(* Logix 5000 project; controller SX_V040001_C001 vendor 1 type 14 code 77 rev 16.23; software revision 16.04; part 2 of 35 *)
(* tags used below, declared in another part *)
   ALARM_BITS : INT[10];
   ALL_KINDS : INT[90];
   Basic : INT;
   CMD : INT[36];
   DRIVE : INT[32];
   EMPTYING : INT[18];
   FP_ALARM_RESET : BOOL;
   G_DInput : DINT[3];
   G_DOutput : DINT[3];
   loading : INT[19];
   louvre : INT[11];
   m_alarm_exist : BOOL;
   m_alarm_horn : BOOL;
   m_element_fault_reset : BOOL;
   m_notstop : BOOL;
   m_on_off_line : BOOL;
   m_power_up : BOOL;
   METERING : INT[44];
   mw_major_fault : DINT;
   PARAMETER : INT[501];
   T_MAX_CURRENT : TIMER;
   T_SCRAPER : TIMER;
   T_START_ALARM : TIMER;
   TEMP : INT[14];
   Z15 : COUNTER;
   Z16 : COUNTER;
   Z17 : COUNTER;
   Z18 : COUNTER;
   Z19 : COUNTER;
   Z20 : COUNTER;
   Z21 : COUNTER;
   Z22 : COUNTER;
   Z23 : COUNTER;
   Z24 : COUNTER;
   Z25 : COUNTER;
   Z26 : COUNTER;
   Z27 : COUNTER;
   Z28 : COUNTER;
   Z29 : COUNTER;
   Z30 : COUNTER;
   Z31 : COUNTER;
   Z32 : COUNTER;
   Z33 : COUNTER;
   Z34 : COUNTER;
   Z35 : COUNTER;
   Z36 : COUNTER;
   Z37 : COUNTER;
   Z38 : COUNTER;
   Z39 : COUNTER;
   Z40 : COUNTER;
   Z41 : COUNTER;
   Z42 : COUNTER;
   Z43 : COUNTER;
   Z44 : COUNTER;
   Z45 : COUNTER;
   Z46 : COUNTER;
   Z47 : COUNTER;
   Z48 : COUNTER;
   Z49 : COUNTER;
   Z50 : COUNTER;
(* MainProgram, continued *)

ROUTINE Alarms   (* ladder *)
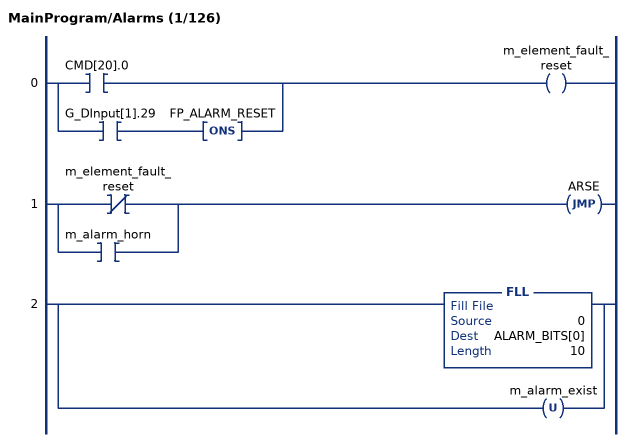
   0: [XIC(CMD[20].0) ,XIC(G_DInput[1].29) ONS(FP_ALARM_RESET) ]OTE(m_element_fault_reset);
   1: [XIO(m_element_fault_reset) ,XIC(m_alarm_horn) ]JMP(ARSE);
   2: [FLL(0,ALARM_BITS[0],10) ,OTU(m_alarm_exist) ];
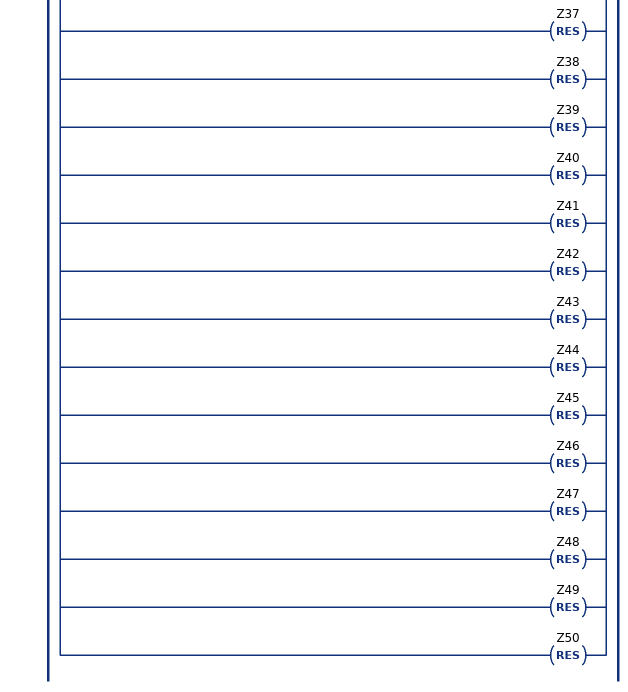
   3: [RES(Z15) ,RES(Z16) ,RES(Z17) ,RES(Z18) ,RES(Z19) ,RES(Z20) ,RES(Z21) ,RES(Z22) ,RES(Z23) ,RES(Z24) ,RES(Z25) ,RES(Z26) ,RES(Z27) ,RES(Z28) ,RES(Z29) ,RES(Z30) ,RES(Z31) ,RES(Z32) ,RES(Z33) ,RES(Z34) ,RES(Z35) ,RES(Z36) ,RES(Z37) ,RES(Z38) ,RES(Z39) ,RES(Z40) ,RES(Z41) ,RES(Z42) ,RES(Z43) ,RES(Z44) ,RES(Z45) ,RES(Z46) ,RES(Z47) ,RES(Z48) ,RES(Z49) ,RES(Z50) ];
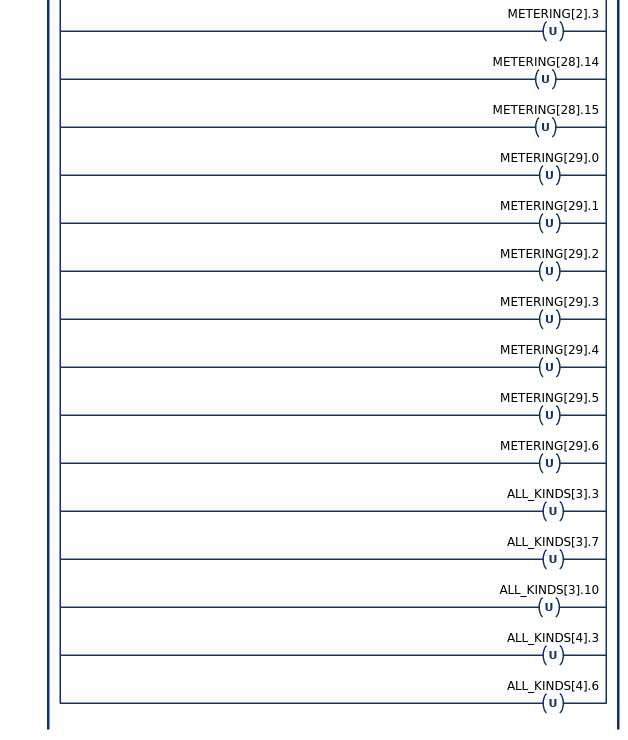
   4: [OTU(TEMP[1].0) ,OTU(TEMP[1].1) ,OTU(TEMP[1].3) ,OTU(TEMP[1].5) ,OTU(TEMP[1].6) ,OTU(DRIVE[2].8) ,OTU(DRIVE[2].9) ,OTU(DRIVE[2].10) ,OTU(DRIVE[2].11) ,OTU(EMPTYING[1].5) ,OTU(EMPTYING[1].7) ,OTU(EMPTYING[1].8) ,OTU(EMPTYING[1].11) ,OTU(EMPTYING[1].12) ,OTU(loading[2].0) ,OTU(loading[2].1) ,OTU(louvre[3].10) ,OTU(louvre[4].10) ,OTU(METERING[1].15) ,OTU(METERING[2].0) ,OTU(METERING[2].1) ,OTU(METERING[2].2) ,OTU(METERING[2].3) ,OTU(METERING[28].14) ,OTU(METERING[28].15) ,OTU(METERING[29].0) ,OTU(METERING[29].1) ,OTU(METERING[29].2) ,OTU(METERING[29].3) ,OTU(METERING[29].4) ,OTU(METERING[29].5) ,OTU(METERING[29].6) ,OTU(ALL_KINDS[3].3) ,OTU(ALL_KINDS[3].7) ,OTU(ALL_KINDS[3].10) ,OTU(ALL_KINDS[4].3) ,OTU(ALL_KINDS[4].6) ];
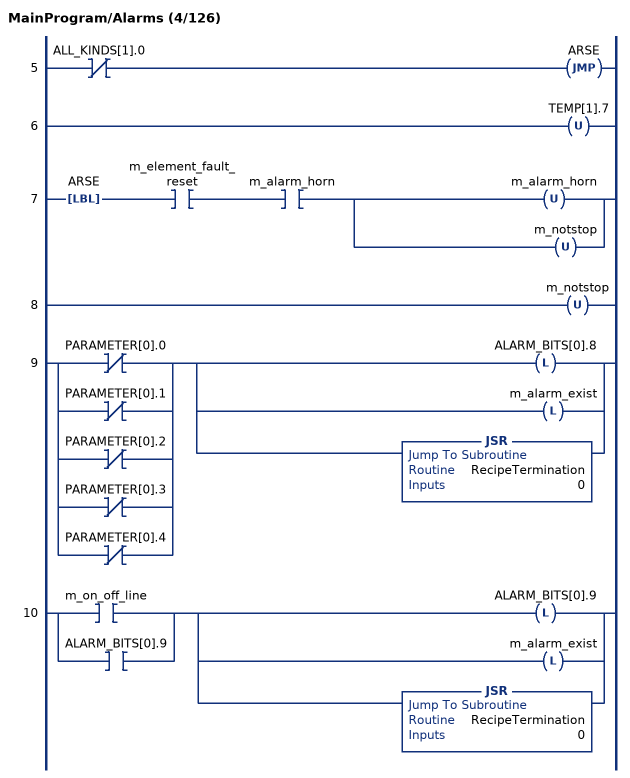
   5: XIO(ALL_KINDS[1].0)JMP(ARSE);
   6: OTU(TEMP[1].7);
   7: LBL(ARSE)XIC(m_element_fault_reset)XIC(m_alarm_horn)[OTU(m_alarm_horn) ,OTU(m_notstop) ];
   8: OTU(m_notstop);
   9: [XIO(PARAMETER[0].0) ,XIO(PARAMETER[0].1) ,XIO(PARAMETER[0].2) ,XIO(PARAMETER[0].3) ,XIO(PARAMETER[0].4) ][OTL(ALARM_BITS[0].8) ,OTL(m_alarm_exist) ,JSR(RecipeTermination,0) ];
   10: [XIC(m_on_off_line) ,XIC(ALARM_BITS[0].9) ][OTL(ALARM_BITS[0].9) ,OTL(m_alarm_exist) ,JSR(RecipeTermination,0) ];
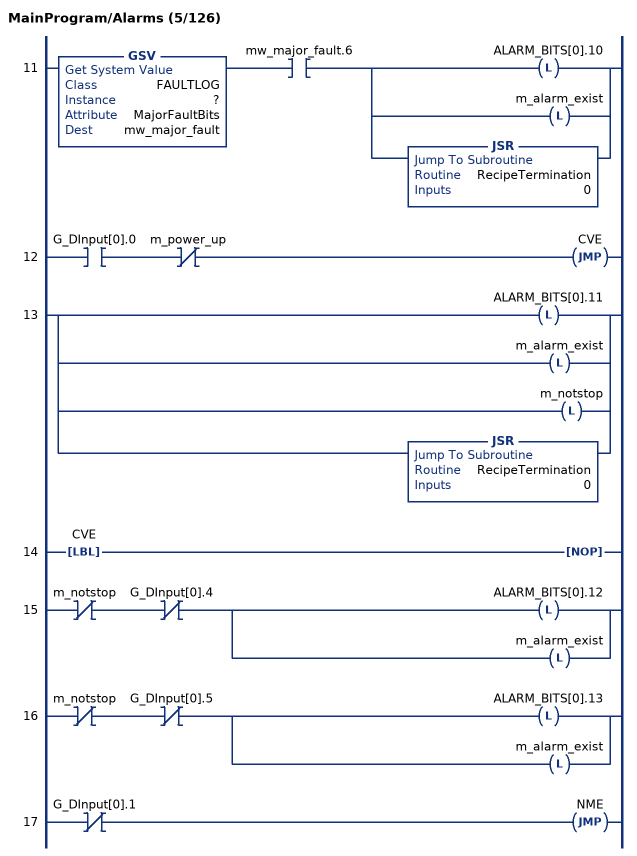
   11: GSV(FAULTLOG,?,MajorFaultBits,mw_major_fault)XIC(mw_major_fault.6)[OTL(ALARM_BITS[0].10) ,OTL(m_alarm_exist) ,JSR(RecipeTermination,0) ];
   12: XIC(G_DInput[0].0)XIO(m_power_up)JMP(CVE);
   13: [OTL(ALARM_BITS[0].11) ,OTL(m_alarm_exist) ,OTL(m_notstop) ,JSR(RecipeTermination,0) ];
   14: LBL(CVE)NOP();
   15: XIO(m_notstop)XIO(G_DInput[0].4)[OTL(ALARM_BITS[0].12) ,OTL(m_alarm_exist) ];
   16: XIO(m_notstop)XIO(G_DInput[0].5)[OTL(ALARM_BITS[0].13) ,OTL(m_alarm_exist) ];
   17: XIO(G_DInput[0].1)JMP(NME);
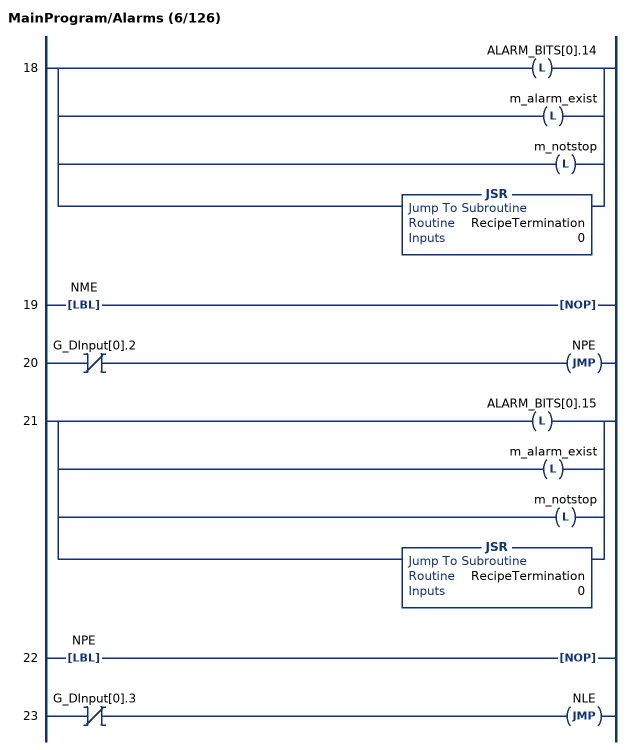
   18: [OTL(ALARM_BITS[0].14) ,OTL(m_alarm_exist) ,OTL(m_notstop) ,JSR(RecipeTermination,0) ];
   19: LBL(NME)NOP();
   20: XIO(G_DInput[0].2)JMP(NPE);
   21: [OTL(ALARM_BITS[0].15) ,OTL(m_alarm_exist) ,OTL(m_notstop) ,JSR(RecipeTermination,0) ];
   22: LBL(NPE)NOP();
   23: XIO(G_DInput[0].3)JMP(NLE);
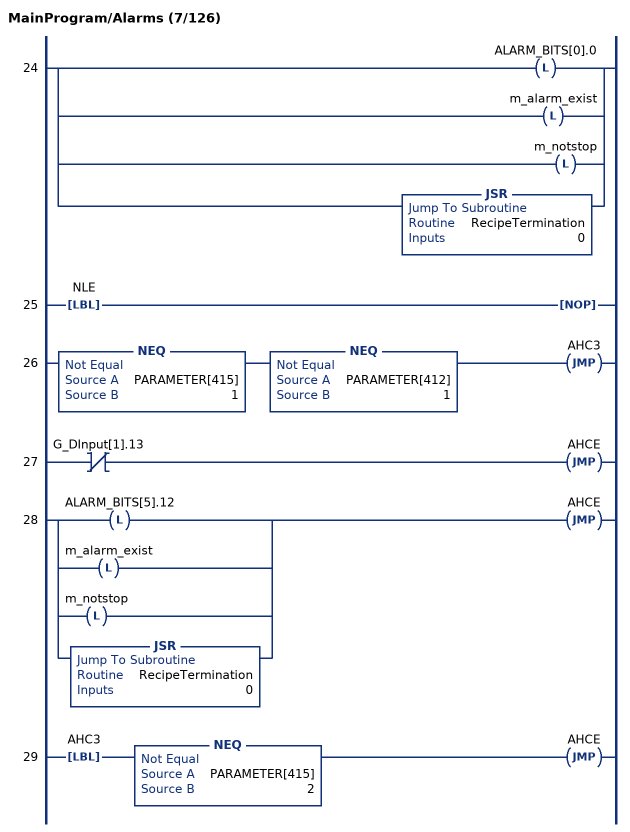
   24: [OTL(ALARM_BITS[0].0) ,OTL(m_alarm_exist) ,OTL(m_notstop) ,JSR(RecipeTermination,0) ];
   25: LBL(NLE)NOP();
   26: NEQ(PARAMETER[415],1)NEQ(PARAMETER[412],1)JMP(AHC3);
   27: XIO(G_DInput[1].13)JMP(AHCE);
   28: [OTL(ALARM_BITS[5].12) ,OTL(m_alarm_exist) ,OTL(m_notstop) ,JSR(RecipeTermination,0) ]JMP(AHCE);
   29: LBL(AHC3)NEQ(PARAMETER[415],2)JMP(AHCE);
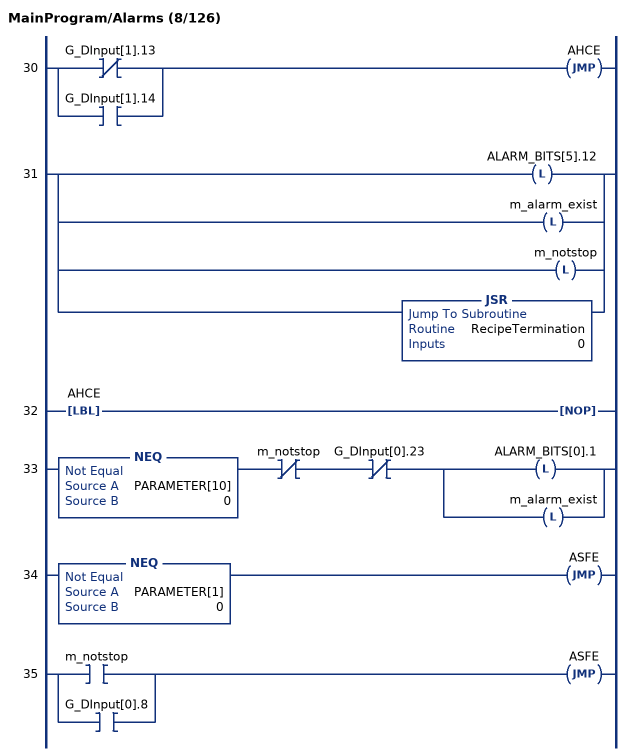
   30: [XIO(G_DInput[1].13) ,XIC(G_DInput[1].14) ]JMP(AHCE);
   31: [OTL(ALARM_BITS[5].12) ,OTL(m_alarm_exist) ,OTL(m_notstop) ,JSR(RecipeTermination,0) ];
   32: LBL(AHCE)NOP();
   33: NEQ(PARAMETER[10],0)XIO(m_notstop)XIO(G_DInput[0].23)[OTL(ALARM_BITS[0].1) ,OTL(m_alarm_exist) ];
   34: NEQ(PARAMETER[1],0)JMP(ASFE);
   35: [XIC(m_notstop) ,XIC(G_DInput[0].8) ]JMP(ASFE);
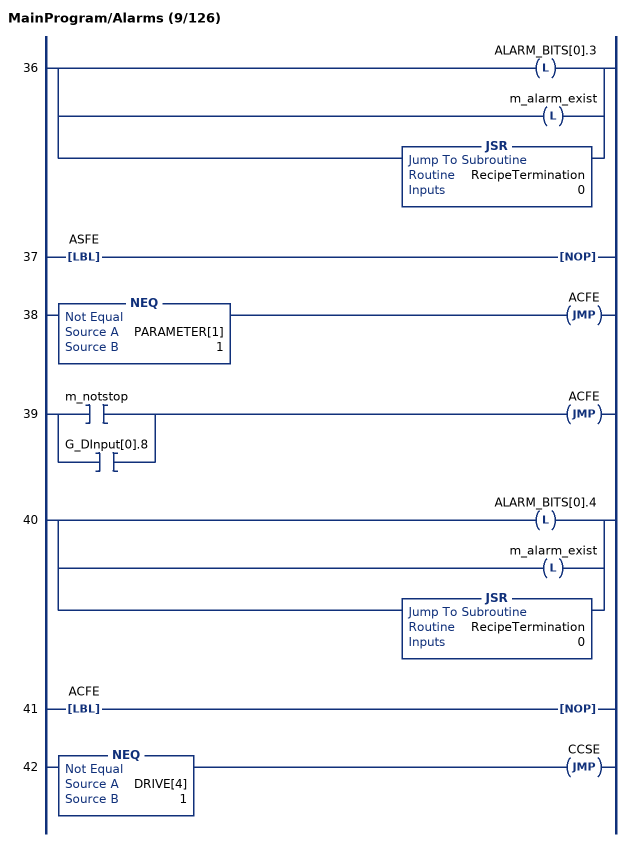
   36: [OTL(ALARM_BITS[0].3) ,OTL(m_alarm_exist) ,JSR(RecipeTermination,0) ];
   37: LBL(ASFE)NOP();
   38: NEQ(PARAMETER[1],1)JMP(ACFE);
   39: [XIC(m_notstop) ,XIC(G_DInput[0].8) ]JMP(ACFE);
   40: [OTL(ALARM_BITS[0].4) ,OTL(m_alarm_exist) ,JSR(RecipeTermination,0) ];
   41: LBL(ACFE)NOP();
   42: NEQ(DRIVE[4],1)JMP(CCSE);
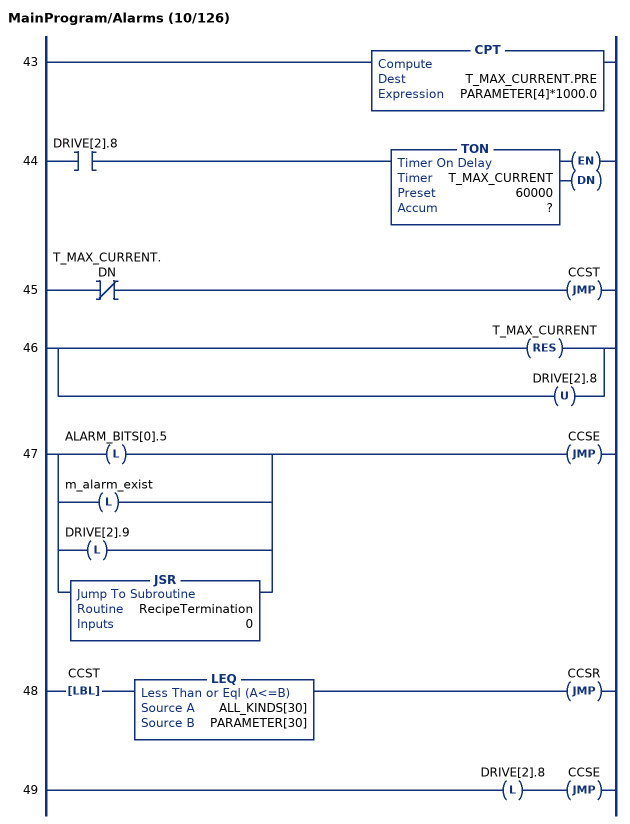
   43: CPT(T_MAX_CURRENT.PRE,PARAMETER[4]*1000.0);
   44: XIC(DRIVE[2].8)TON(T_MAX_CURRENT,?,?);
   45: XIO(T_MAX_CURRENT.DN)JMP(CCST);
   46: [RES(T_MAX_CURRENT) ,OTU(DRIVE[2].8) ];
   47: [OTL(ALARM_BITS[0].5) ,OTL(m_alarm_exist) ,OTL(DRIVE[2].9) ,JSR(RecipeTermination,0) ]JMP(CCSE);
   48: LBL(CCST)LEQ(ALL_KINDS[30],PARAMETER[30])JMP(CCSR);
   49: OTL(DRIVE[2].8)JMP(CCSE);
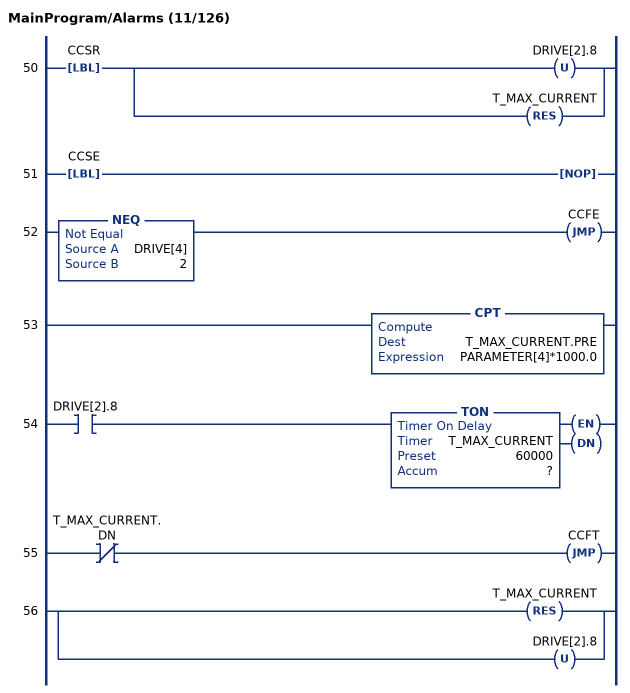
   50: LBL(CCSR)[OTU(DRIVE[2].8) ,RES(T_MAX_CURRENT) ];
   51: LBL(CCSE)NOP();
   52: NEQ(DRIVE[4],2)JMP(CCFE);
   53: CPT(T_MAX_CURRENT.PRE,PARAMETER[4]*1000.0);
   54: XIC(DRIVE[2].8)TON(T_MAX_CURRENT,?,?);
   55: XIO(T_MAX_CURRENT.DN)JMP(CCFT);
   56: [RES(T_MAX_CURRENT) ,OTU(DRIVE[2].8) ];
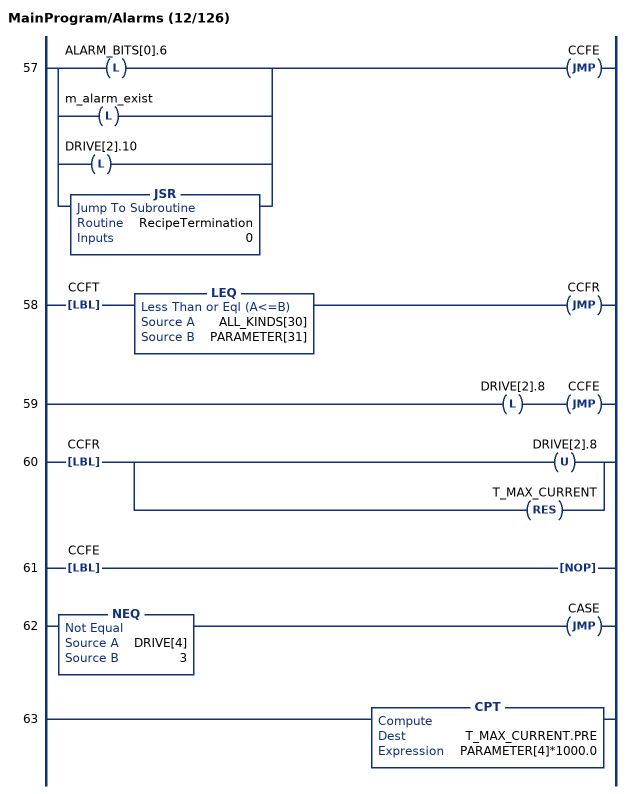
   57: [OTL(ALARM_BITS[0].6) ,OTL(m_alarm_exist) ,OTL(DRIVE[2].10) ,JSR(RecipeTermination,0) ]JMP(CCFE);
   58: LBL(CCFT)LEQ(ALL_KINDS[30],PARAMETER[31])JMP(CCFR);
   59: OTL(DRIVE[2].8)JMP(CCFE);
   60: LBL(CCFR)[OTU(DRIVE[2].8) ,RES(T_MAX_CURRENT) ];
   61: LBL(CCFE)NOP();
   62: NEQ(DRIVE[4],3)JMP(CASE);
   63: CPT(T_MAX_CURRENT.PRE,PARAMETER[4]*1000.0);
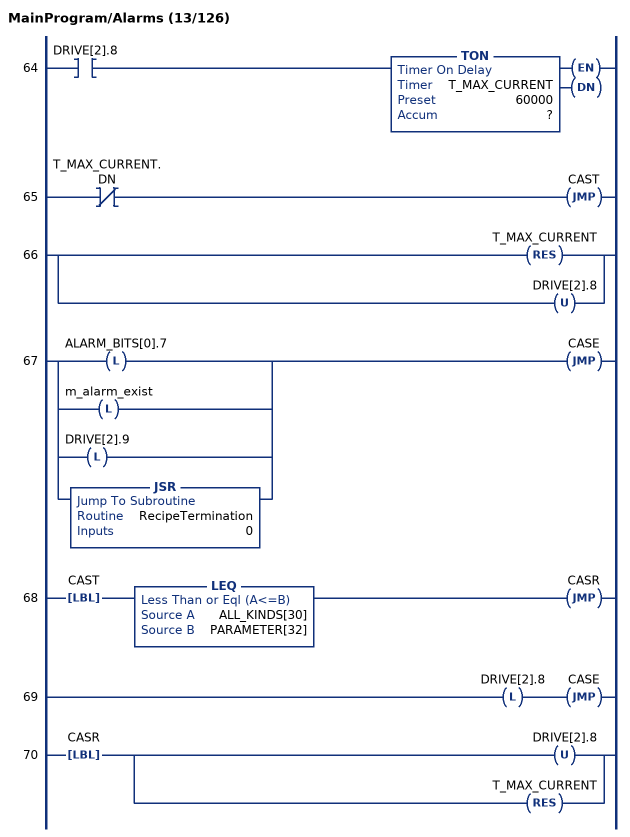
   64: XIC(DRIVE[2].8)TON(T_MAX_CURRENT,?,?);
   65: XIO(T_MAX_CURRENT.DN)JMP(CAST);
   66: [RES(T_MAX_CURRENT) ,OTU(DRIVE[2].8) ];
   67: [OTL(ALARM_BITS[0].7) ,OTL(m_alarm_exist) ,OTL(DRIVE[2].9) ,JSR(RecipeTermination,0) ]JMP(CASE);
   68: LBL(CAST)LEQ(ALL_KINDS[30],PARAMETER[32])JMP(CASR);
   69: OTL(DRIVE[2].8)JMP(CASE);
   70: LBL(CASR)[OTU(DRIVE[2].8) ,RES(T_MAX_CURRENT) ];
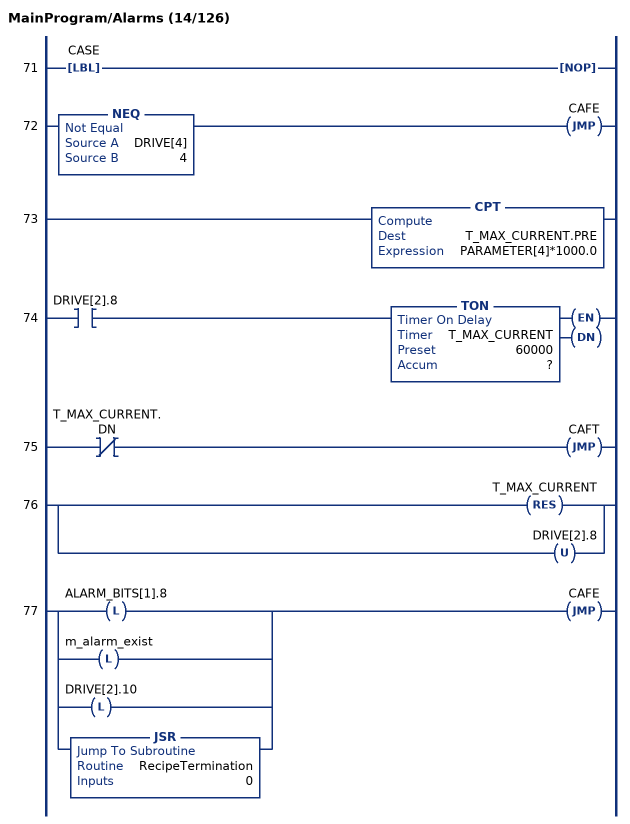
   71: LBL(CASE)NOP();
   72: NEQ(DRIVE[4],4)JMP(CAFE);
   73: CPT(T_MAX_CURRENT.PRE,PARAMETER[4]*1000.0);
   74: XIC(DRIVE[2].8)TON(T_MAX_CURRENT,?,?);
   75: XIO(T_MAX_CURRENT.DN)JMP(CAFT);
   76: [RES(T_MAX_CURRENT) ,OTU(DRIVE[2].8) ];
   77: [OTL(ALARM_BITS[1].8) ,OTL(m_alarm_exist) ,OTL(DRIVE[2].10) ,JSR(RecipeTermination,0) ]JMP(CAFE);
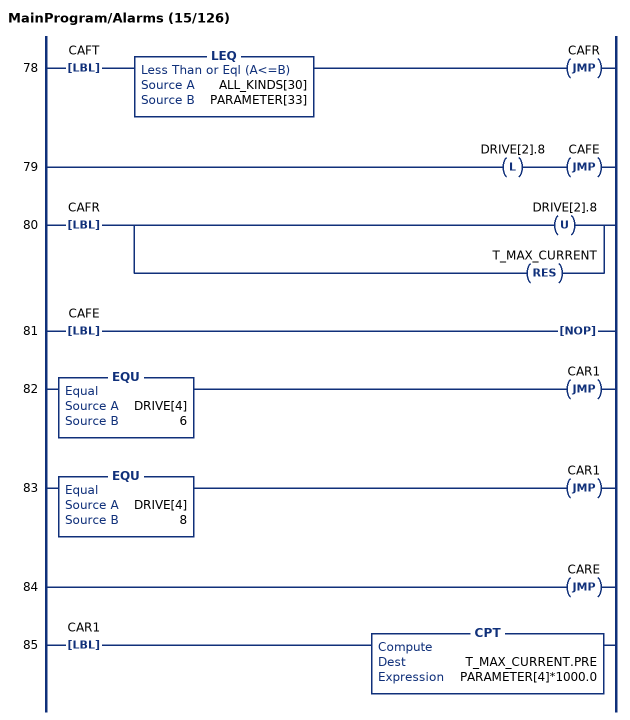
   78: LBL(CAFT)LEQ(ALL_KINDS[30],PARAMETER[33])JMP(CAFR);
   79: OTL(DRIVE[2].8)JMP(CAFE);
   80: LBL(CAFR)[OTU(DRIVE[2].8) ,RES(T_MAX_CURRENT) ];
   81: LBL(CAFE)NOP();
   82: EQU(DRIVE[4],6)JMP(CAR1);
   83: EQU(DRIVE[4],8)JMP(CAR1);
   84: JMP(CARE);
   85: LBL(CAR1)CPT(T_MAX_CURRENT.PRE,PARAMETER[4]*1000.0);
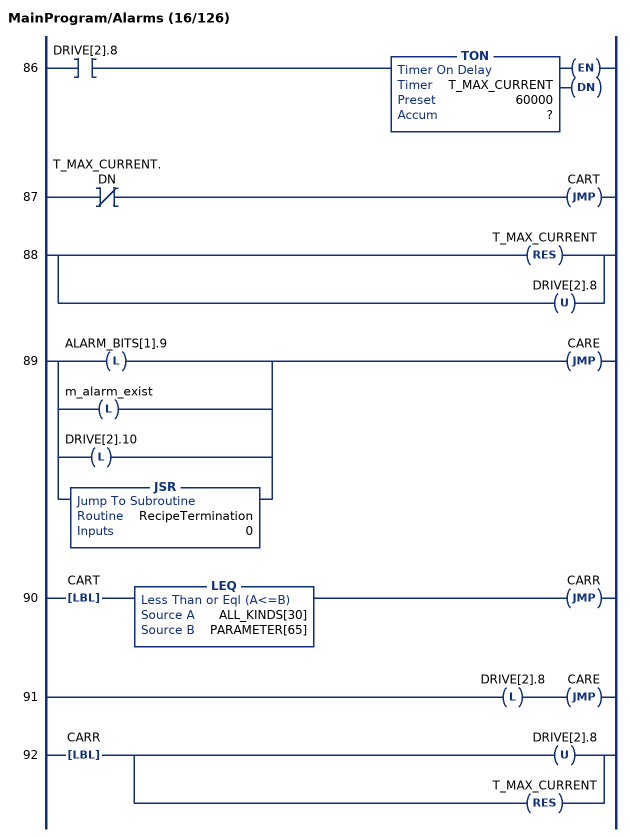
   86: XIC(DRIVE[2].8)TON(T_MAX_CURRENT,?,?);
   87: XIO(T_MAX_CURRENT.DN)JMP(CART);
   88: [RES(T_MAX_CURRENT) ,OTU(DRIVE[2].8) ];
   89: [OTL(ALARM_BITS[1].9) ,OTL(m_alarm_exist) ,OTL(DRIVE[2].10) ,JSR(RecipeTermination,0) ]JMP(CARE);
   90: LBL(CART)LEQ(ALL_KINDS[30],PARAMETER[65])JMP(CARR);
   91: OTL(DRIVE[2].8)JMP(CARE);
   92: LBL(CARR)[OTU(DRIVE[2].8) ,RES(T_MAX_CURRENT) ];
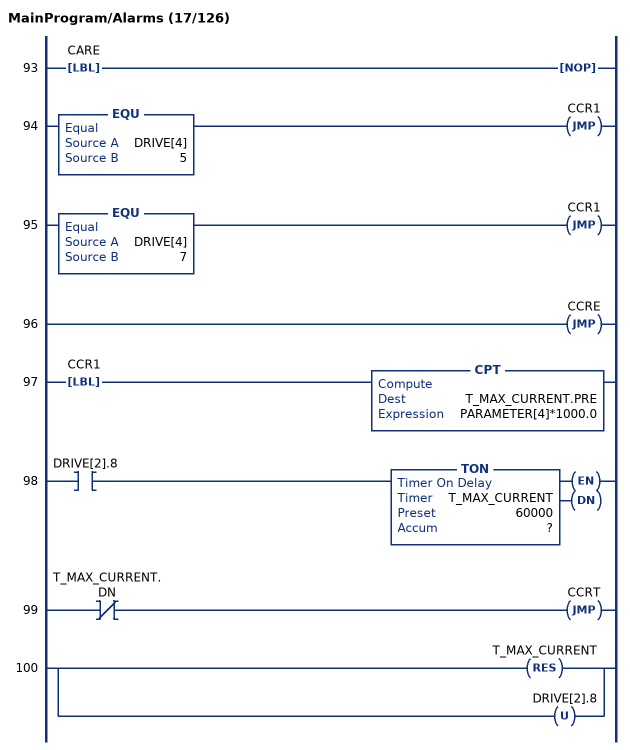
   93: LBL(CARE)NOP();
   94: EQU(DRIVE[4],5)JMP(CCR1);
   95: EQU(DRIVE[4],7)JMP(CCR1);
   96: JMP(CCRE);
   97: LBL(CCR1)CPT(T_MAX_CURRENT.PRE,PARAMETER[4]*1000.0);
   98: XIC(DRIVE[2].8)TON(T_MAX_CURRENT,?,?);
   99: XIO(T_MAX_CURRENT.DN)JMP(CCRT);
   100: [RES(T_MAX_CURRENT) ,OTU(DRIVE[2].8) ];
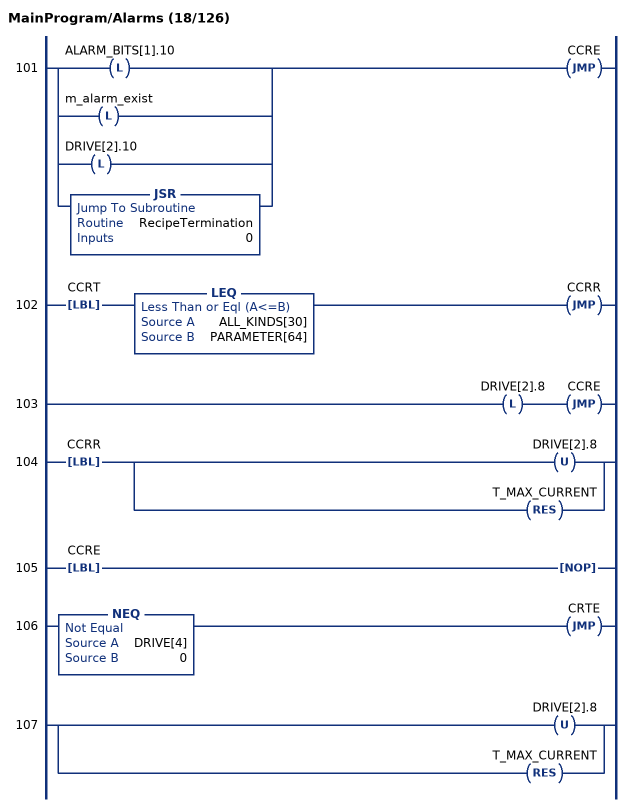
   101: [OTL(ALARM_BITS[1].10) ,OTL(m_alarm_exist) ,OTL(DRIVE[2].10) ,JSR(RecipeTermination,0) ]JMP(CCRE);
   102: LBL(CCRT)LEQ(ALL_KINDS[30],PARAMETER[64])JMP(CCRR);
   103: OTL(DRIVE[2].8)JMP(CCRE);
   104: LBL(CCRR)[OTU(DRIVE[2].8) ,RES(T_MAX_CURRENT) ];
   105: LBL(CCRE)NOP();
   106: NEQ(DRIVE[4],0)JMP(CRTE);
   107: [OTU(DRIVE[2].8) ,RES(T_MAX_CURRENT) ];
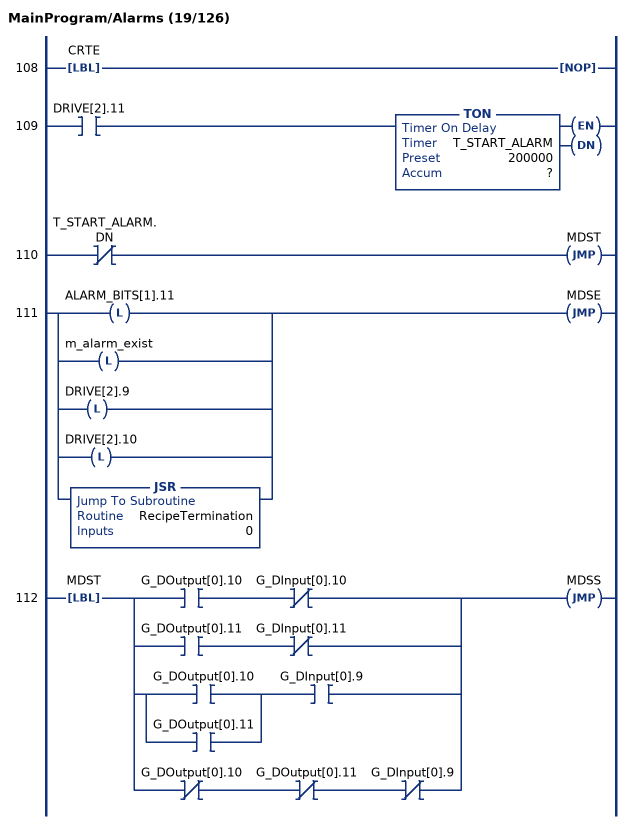
   108: LBL(CRTE)NOP();
   109: XIC(DRIVE[2].11)TON(T_START_ALARM,?,?);
   110: XIO(T_START_ALARM.DN)JMP(MDST);
   111: [OTL(ALARM_BITS[1].11) ,OTL(m_alarm_exist) ,OTL(DRIVE[2].9) ,OTL(DRIVE[2].10) ,JSR(RecipeTermination,0) ]JMP(MDSE);
   112: LBL(MDST)[XIC(G_DOutput[0].10) XIO(G_DInput[0].10) ,XIC(G_DOutput[0].11) XIO(G_DInput[0].11) ,[XIC(G_DOutput[0].10) ,XIC(G_DOutput[0].11) ] XIC(G_DInput[0].9) ,XIO(G_DOutput[0].10) XIO(G_DOutput[0].11) XIO(G_DInput[0].9) ]JMP(MDSS);
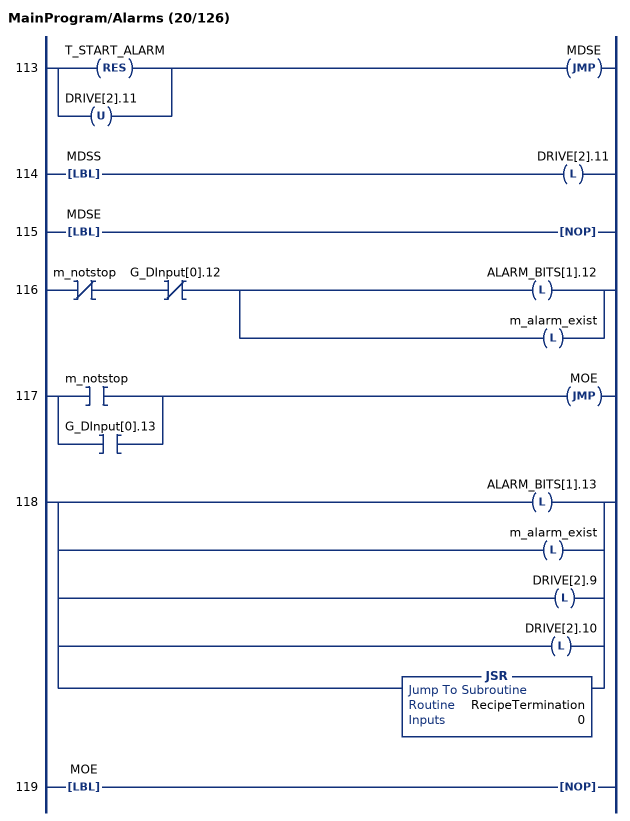
   113: [RES(T_START_ALARM) ,OTU(DRIVE[2].11) ]JMP(MDSE);
   114: LBL(MDSS)OTL(DRIVE[2].11);
   115: LBL(MDSE)NOP();
   116: XIO(m_notstop)XIO(G_DInput[0].12)[OTL(ALARM_BITS[1].12) ,OTL(m_alarm_exist) ];
   117: [XIC(m_notstop) ,XIC(G_DInput[0].13) ]JMP(MOE);
   118: [OTL(ALARM_BITS[1].13) ,OTL(m_alarm_exist) ,OTL(DRIVE[2].9) ,OTL(DRIVE[2].10) ,JSR(RecipeTermination,0) ];
   119: LBL(MOE)NOP();
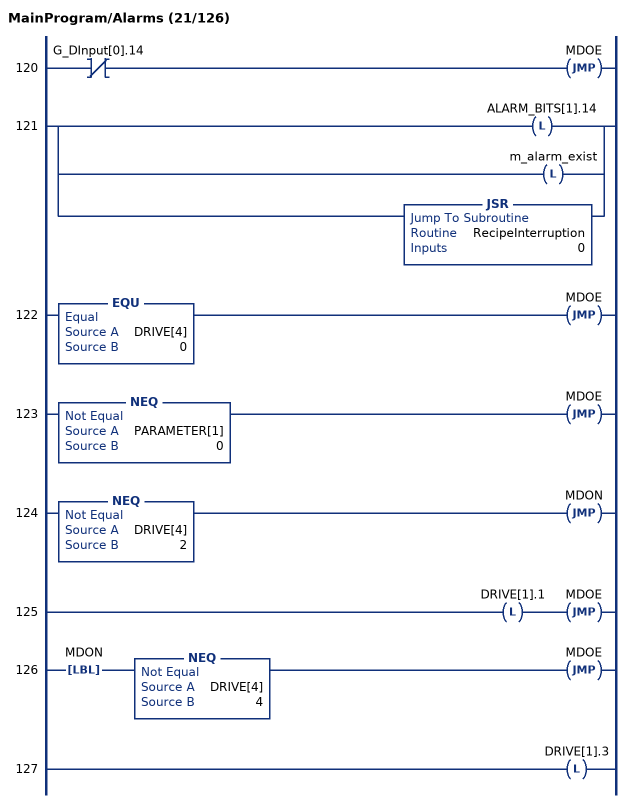
   120: XIO(G_DInput[0].14)JMP(MDOE);
   121: [OTL(ALARM_BITS[1].14) ,OTL(m_alarm_exist) ,JSR(RecipeInterruption,0) ];
   122: EQU(DRIVE[4],0)JMP(MDOE);
   123: NEQ(PARAMETER[1],0)JMP(MDOE);
   124: NEQ(DRIVE[4],2)JMP(MDON);
   125: OTL(DRIVE[1].1)JMP(MDOE);
   126: LBL(MDON)NEQ(DRIVE[4],4)JMP(MDOE);
   127: OTL(DRIVE[1].3);
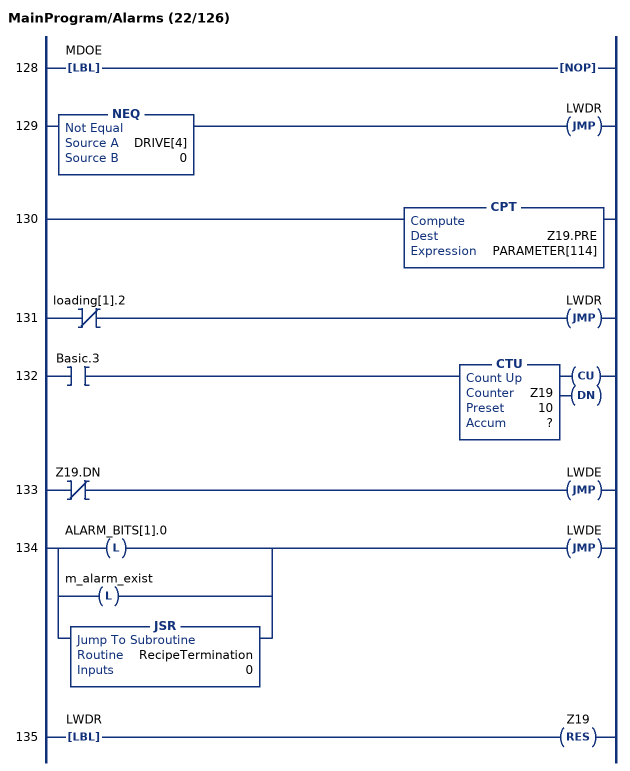
   128: LBL(MDOE)NOP();
   129: NEQ(DRIVE[4],0)JMP(LWDR);
   130: CPT(Z19.PRE,PARAMETER[114]);
   131: XIO(loading[1].2)JMP(LWDR);
   132: XIC(Basic.3)CTU(Z19,?,?);
   133: XIO(Z19.DN)JMP(LWDE);
   134: [OTL(ALARM_BITS[1].0) ,OTL(m_alarm_exist) ,JSR(RecipeTermination,0) ]JMP(LWDE);
   135: LBL(LWDR)RES(Z19);
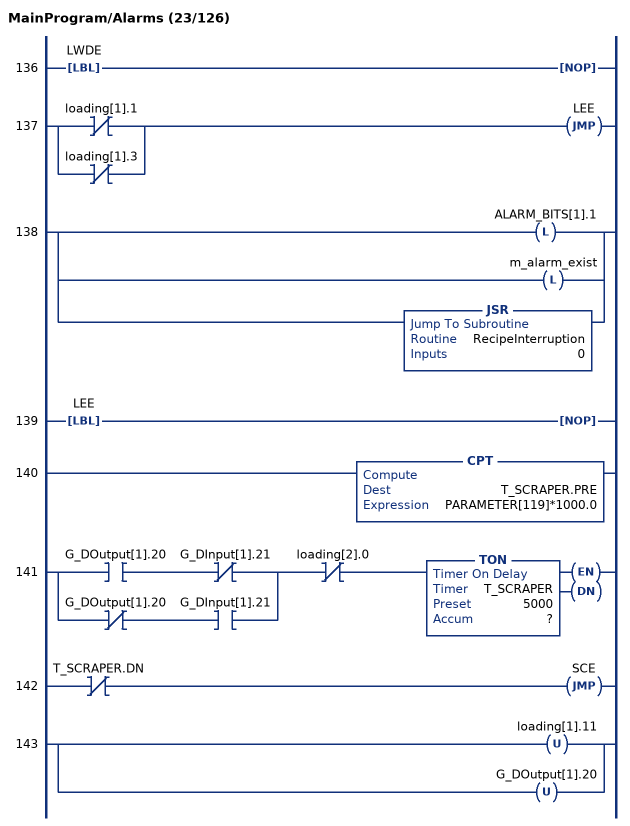
   136: LBL(LWDE)NOP();
   137: [XIO(loading[1].1) ,XIO(loading[1].3) ]JMP(LEE);
   138: [OTL(ALARM_BITS[1].1) ,OTL(m_alarm_exist) ,JSR(RecipeInterruption,0) ];
   139: LBL(LEE)NOP();
   140: CPT(T_SCRAPER.PRE,PARAMETER[119]*1000.0);
   141: [XIC(G_DOutput[1].20) XIO(G_DInput[1].21) ,XIO(G_DOutput[1].20) XIC(G_DInput[1].21) ]XIO(loading[2].0)TON(T_SCRAPER,?,?);
   142: XIO(T_SCRAPER.DN)JMP(SCE);
   143: [OTU(loading[1].11) ,OTU(G_DOutput[1].20) ];
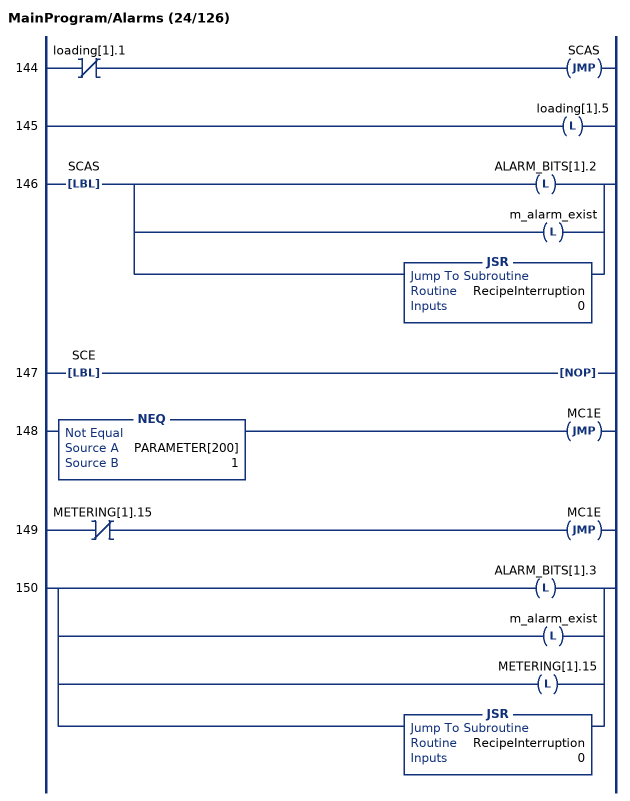
   144: XIO(loading[1].1)JMP(SCAS);
   145: OTL(loading[1].5);
   146: LBL(SCAS)[OTL(ALARM_BITS[1].2) ,OTL(m_alarm_exist) ,JSR(RecipeInterruption,0) ];
   147: LBL(SCE)NOP();
   148: NEQ(PARAMETER[200],1)JMP(MC1E);
   149: XIO(METERING[1].15)JMP(MC1E);
   150: [OTL(ALARM_BITS[1].3) ,OTL(m_alarm_exist) ,OTL(METERING[1].15) ,JSR(RecipeInterruption,0) ];
